{attribute addProperty BoxType "ELM9410-0000-0018"}
{attribute addProperty Id "MMS_Device_InputsAT %I*MMS_Device_Inputs_840DB41B810MMS_Acceleration_StatusAT %I*MMS_Acceleration_Status_2FF1A4723240MMS_Acceleration_X_AxisAT %I*MMS_Acceleration_X_Axis_2EF51F001620MMS_Acceleration_Y_AxisAT %I*MMS_Acceleration_Y_Axis_2EF51F001620MMS_Acceleration_Z_AxisAT %I*MMS_Acceleration_Z_Axis_2EF51F001620MMS_Acceleration_TimestampAT %I*MMS_Acceleration_Timestamp_0B25C1A46480MMS_Voltage_Us_In_InputsAT %I*MMS_Voltage_Us_In_Inputs_BF33E0C16480MMS_Voltage_Up_In_InputsAT %I*MMS_Voltage_Up_In_Inputs_BF33E0C16480MMS_Voltage_Up_Out_InputsAT %I*MMS_Voltage_Up_Out_Inputs_BF33E0C16480MMS_Device_OutputsAT %Q*MMS_Device_Outputs_39C15ABC1620WcStateAT %I*WcState_F855686C1620InfoDataAT %I*InfoData_0BDED7BF144180"}
{attribute addProperty CRC "970172899"}
{attribute addProperty SizeInBites "520"}
{attribute addProperty SizeInBytes "65"}
TYPE ELM9410_75EA563B :
STRUCT
	{attribute addProperty Name "MMS_Device_Inputs"}
	MMS_Device_Inputs : MMS_Device_Inputs_840DB41B;
	{attribute addProperty Name "MMS_Acceleration_Status"}
	MMS_Acceleration_Status : MMS_Acceleration_Status_2FF1A472;
	{attribute addProperty Name "MMS_Acceleration_X_Axis"}
	MMS_Acceleration_X_Axis : MMS_Acceleration_X_Axis_2EF51F00;
	{attribute addProperty Name "MMS_Acceleration_Y_Axis"}
	MMS_Acceleration_Y_Axis : MMS_Acceleration_Y_Axis_2EF51F00;
	{attribute addProperty Name "MMS_Acceleration_Z_Axis"}
	MMS_Acceleration_Z_Axis : MMS_Acceleration_Z_Axis_2EF51F00;
	{attribute addProperty Name "MMS_Acceleration_Timestamp"}
	MMS_Acceleration_Timestamp : MMS_Acceleration_Timestamp_0B25C1A4;
	{attribute addProperty Name "MMS_Voltage_Us_In_Inputs"}
	MMS_Voltage_Us_In_Inputs : MMS_Voltage_Us_In_Inputs_BF33E0C1;
	{attribute addProperty Name "MMS_Voltage_Up_In_Inputs"}
	MMS_Voltage_Up_In_Inputs : MMS_Voltage_Up_In_Inputs_BF33E0C1;
	{attribute addProperty Name "MMS_Voltage_Up_Out_Inputs"}
	MMS_Voltage_Up_Out_Inputs : MMS_Voltage_Up_Out_Inputs_BF33E0C1;
	{attribute addProperty Name "MMS_Device_Outputs"}
	MMS_Device_Outputs : MMS_Device_Outputs_39C15ABC;
	{attribute addProperty Name "WcState"}
	WcState : WcState_F855686C;
	{attribute addProperty Name "InfoData"}
	InfoData : InfoData_0BDED7BF;
END_STRUCT
END_TYPE

(* stored: Version 1.2.0.0, ProductVersion 3.1.4024.9
   DUT ELM9410_75EA563B: Id {2dc4d34d-df2d-4af6-9658-5d1866670125} *)
